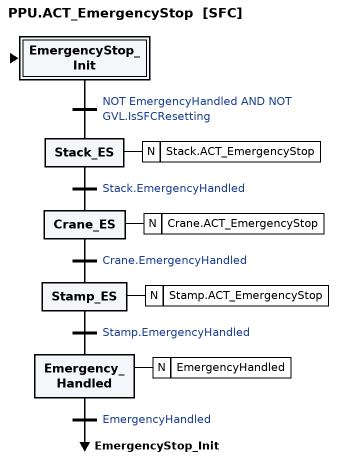
(* [picture p24: PPU.ACT_EmergencyStop, SFC] *)
INITIAL_STEP EmergencyStop_Init:
END_STEP
TRANSITION FROM EmergencyStop_Init TO Stack_ES
  := NOT EmergencyHandled AND NOT GVL.IsSFCResetting;
END_TRANSITION
STEP Stack_ES:
  Stack.ACT_EmergencyStop(N);
END_STEP
TRANSITION FROM Stack_ES TO Crane_ES
  := Stack.EmergencyHandled;
END_TRANSITION
STEP Crane_ES:
  Crane.ACT_EmergencyStop(N);
END_STEP
TRANSITION FROM Crane_ES TO Stamp_ES
  := Crane.EmergencyHandled;
END_TRANSITION
STEP Stamp_ES:
  Stamp.ACT_EmergencyStop(N);
END_STEP
TRANSITION FROM Stamp_ES TO Emergency_Handled
  := Stamp.EmergencyHandled;
END_TRANSITION
STEP Emergency_Handled:
  EmergencyHandled(N);
END_STEP
TRANSITION FROM Emergency_Handled TO EmergencyStop_Init
  := EmergencyHandled;
END_TRANSITION
END_ACTION

ACTION ACT_Init:
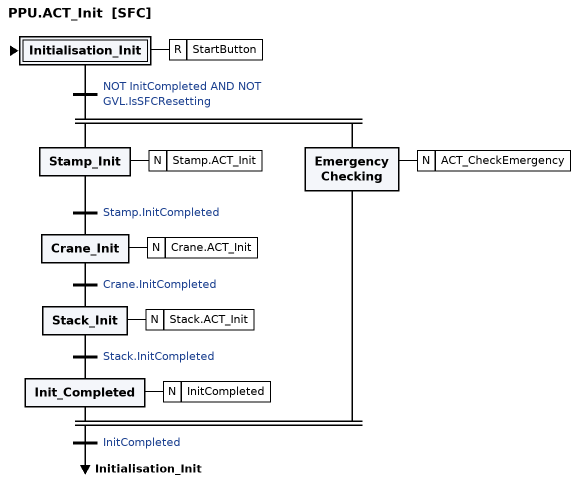
INITIAL_STEP Initialisation_Init:
  StartButton(R);
END_STEP
TRANSITION FROM Initialisation_Init TO (Stamp_Init, EmergencyChecking)
  := NOT InitCompleted AND NOT GVL.IsSFCResetting;
END_TRANSITION
STEP Stamp_Init:
  Stamp.ACT_Init(N);
END_STEP
TRANSITION FROM Stamp_Init TO Crane_Init
  := Stamp.InitCompleted;
END_TRANSITION
STEP Crane_Init:
  Crane.ACT_Init(N);
END_STEP
TRANSITION FROM Crane_Init TO Stack_Init
  := Crane.InitCompleted;
END_TRANSITION
STEP Stack_Init:
  Stack.ACT_Init(N);
END_STEP
TRANSITION FROM Stack_Init TO Init_Completed
  := Stack.InitCompleted;
END_TRANSITION
STEP Init_Completed:
  InitCompleted(N);
END_STEP
TRANSITION FROM (Init_Completed, EmergencyChecking) TO Initialisation_Init
  := InitCompleted;
END_TRANSITION
STEP EmergencyChecking:
  ACT_CheckEmergency(N);
END_STEP
END_ACTION
END_FUNCTION_BLOCK

CONFIGURATION Application
  RESOURCE Scenario_4b ON PLC
(* global variable list GVL *)
{attribute 'qualified_only'}
VAR_GLOBAL
	IsSFCResetting : BOOL;
END_VAR
    TASK PlcTask(INTERVAL := T#0ms, PRIORITY := 20);
    PROGRAM MAIN WITH PlcTask : MAIN;
  END_RESOURCE
END_CONFIGURATION
